(*

.. <legal notes>

legal notes
=================
| SPDX-FileCopyrightText: © 2025 Oleksandr Tiutyk <trofimich@gmail.com>
| SPDX-License-Identifier: LGPL-3.0-only
| For details check: LGPL-3.0-only_

.. _LGPL-3.0-only: https://www.gnu.org/licenses/lgpl-3.0.en.html

.. </legal notes>

*)

{attribute 'no_explicit_call' := 'do not call this POU directly'}
PROGRAM CurrentNamespace
VAR
	_NamespaceExtractor : NamespaceExtractor;
END_VAR

{attribute 'monitoring' := 'call'}
PROPERTY Name : STRING
GET
Name := _NamespaceExtractor.CurrentNamespace;
END_GET
END_PROPERTY

END_PROGRAM

(* stored: Version 1.1.0.1
   POU CurrentNamespace: Id {f24d7c34-d6e3-45a4-9a69-d0c668832c17}, SpecialFunc None
   Property Name: Id {ab92da57-5dc1-4458-91d8-c6f305012951}
   Get Get: Id {768d7488-7081-4761-adfb-5b76040ddcb9} *)
